FUNCTION fc_MODR : real
VAR_INPUT
	IN : REAL;
	DIVI : REAL;
END_VAR
VAR
END_VAR

IF divi = 0.0 THEN
	fc_MODR := 0.0;
ELSE
	fc_MODR := in - DINT_TO_REAL(fc_Floor2(in / divi)) * divi;
END_IF;

END_FUNCTION

(* stored: Version 1.1.0.1, ProductVersion 3.1.4024.11
   POU fc_MODR: Id {783d0025-a7ed-4606-997e-1a2a6d758773}, SpecialFunc None *)
